FUNCTION_BLOCK NewAdapter2 (* Template for an empty basic function block *)
  (* Standard: 61499-2; Description: Copyright (c) 2019 Jan Holzweber This program and the accompanying materials are made available under the terms of the Eclipse Public License 2.0 which is available at https://www.eclipse.org/legal/epl-2.0/ SPDX-License-Identifier: EPL-2.0 *)
  (* Version 1.0, 2019-06-10, Jan Holzweber *)
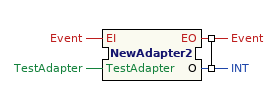
  EVENT_INPUT
    EI;
  END_EVENT
  EVENT_OUTPUT
    EO WITH O;
  END_EVENT
  VAR_OUTPUT
    O : INT;
  END_VAR
  SOCKETS
    TestAdapter : TestAdapter;
  END_SOCKETS
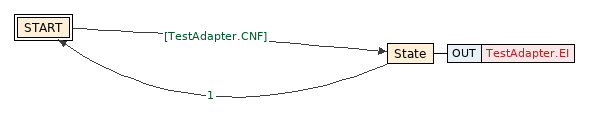
  EC_STATES
    START; (* Initial State *)
    State : OUT -> TestAdapter.EI;
  END_STATES
  EC_TRANSITIONS
    START TO State := [TestAdapter.CNF];
    State TO START := 1;
  END_TRANSITIONS
  ALGORITHM OUT IN ST: (* new algorithm *)
O:= TestAdapter.D0;
TestAdapter.DI:= 1 +D0;
  END_ALGORITHM
END_FUNCTION_BLOCK
